PROGRAM Laser
VAR
	nLaserRawValue 	AT %I* 	: INT := 0;
	nLaserOffset			: INT := 200;
	tmpVal					: INT;
	sLaserError		AT %I*	: BOOL;
END_VAR


IF nLaserRawValue > 16#6C00 THEN
	Module_IO.nLaserValue:= 0;
ELSE
	tmpVal:= (WORD_TO_INT(nLaserRawValue * 4800 / 16#6C00)+ nLaserOffset);
	Module_IO.nLaserValue:= tmpVal;
END_IF

END_PROGRAM

(* stored: Version 1.1.0.1, ProductVersion 3.1.4024.11
   POU Laser: Id {c67e9438-5fda-48d0-a654-0ce65fa0f93f}, SpecialFunc None *)
